// TIA Portal V19 export
TYPE "IO Burkett Type 8691 r3"
   STRUCT
      IN : Struct
         Addr : Int;   // First Byte address of 4 byte address space
         Locate : Bool;   // Rapid Flash LED's
         Activate : Bool;   // Activate pilot valve
      END_STRUCT;
      OUT : Struct
         ValvePosition : Real;   // 0-100%
         NumarState : Byte;   // 0=diagPassive,1=diagActive,2=MaintenanceRequired,3=OutOfSpec,4=warn,5=error
         OperationState : Byte;   // See block comment
         POS2 : Bool;   // True = process valve is in end position defined by activated pilot valve.
         POS1 : Bool;   // True = process valve is in end position defined by deactivated pilot valve.
         EndPositionClose : Bool;   // True = Process Valve is closed.
         EndPositionOpen : Bool;   // True = Process Valve is open.
         O_DI4 : Bool;   // Output signal status Pin 4
         O_DI2 : Bool;   // Output signal status Pin 2
         O_DA : Bool;   // Output device recognised
         O_DE : Bool;   // Output device error event has appeared
         O_PQ : Bool;   // Output port qualifer proces data valid
      END_STRUCT;
      IN_OUT : Struct
         HMI_CMD : Word;
         HMI_INFO : Word;
      END_STRUCT;
   END_STRUCT;
END_TYPE
